// TIA Portal V18 export
FUNCTION "Test" : Void   // FC1, STL
{ S7_Optimized_Access := 'TRUE' }
VERSION : 0.1
// stored: AutoNumber true, UDAEnableTagReadback false
BEGIN

NETWORK
TITLE = 
      NOP   0;

END_FUNCTION
